FUNCTION_BLOCK FB_Blinklicht
VAR_INPUT
	bEinAus		: BOOL;
	tPeriode	: TIME := T#1S;
END_VAR
VAR_OUTPUT
	bBlink		: BOOL;
END_VAR
VAR
	fbTon		: TON;
END_VAR

fbTon(IN:=bEinAus AND NOT fbTon.Q , PT:=tPeriode , Q=> , ET=> );

IF fbTON.ET <= fbTON.PT/2 THEN
	bBlink := FALSE;
ELSE
	bBlink := TRUE;
END_IF

IF NOT bEinAus THEN
	bBlink := FALSE;
END_IF

END_FUNCTION_BLOCK

(* stored: Version 1.1.0.1, ProductVersion 3.1.4024.15
   POU FB_Blinklicht: Id {3afcacf6-06f9-424f-ac1b-d90aa3ff3890}, SpecialFunc None *)
